{attribute addProperty BoxType "KL1644-0050"}
{attribute addProperty Id "Channel_1Channel_7DECC1C800Channel_2Channel_7DECC1C800Channel_3Channel_7DECC1C800Channel_4Channel_7DECC1C800"}
{attribute addProperty CRC "631967696"}
{attribute addProperty SizeInBites "0"}
{attribute addProperty SizeInBytes "0"}
TYPE KL_25AB0FD0 :
STRUCT
	{attribute addProperty Name "Channel_1"}
	Channel_1 : Channel_7DECC1C8;
	{attribute addProperty Name "Channel_2"}
	Channel_2 : Channel_7DECC1C8;
	{attribute addProperty Name "Channel_3"}
	Channel_3 : Channel_7DECC1C8;
	{attribute addProperty Name "Channel_4"}
	Channel_4 : Channel_7DECC1C8;
END_STRUCT
END_TYPE

(* stored: Version 1.2.0.0, ProductVersion 3.1.4024.9
   DUT KL_25AB0FD0: Id {cdddcfed-7761-49c7-b922-9cd062561138} *)
